// An enum to specify the memory area type of an address.
{attribute 'qualified_only'}
{attribute 'to_string'}
TYPE E_AddressMemoryArea :
(
	_ 		:= 0, 	// Unknown/Invalid.
	Static	:= 1, 	// Static memory.
	Dynamic	:= 2, 	// Dynamic memory.
	CNC		:= 3	// CNC static memory.
)BYTE;
END_TYPE

(* stored: Version 1.1.0.1
   EnumerationTextList E_AddressMemoryArea: Id {6aae7e94-3d7e-0a93-3ae5-b637be439f76} *)
